RoboDK station: project robotics.rdk

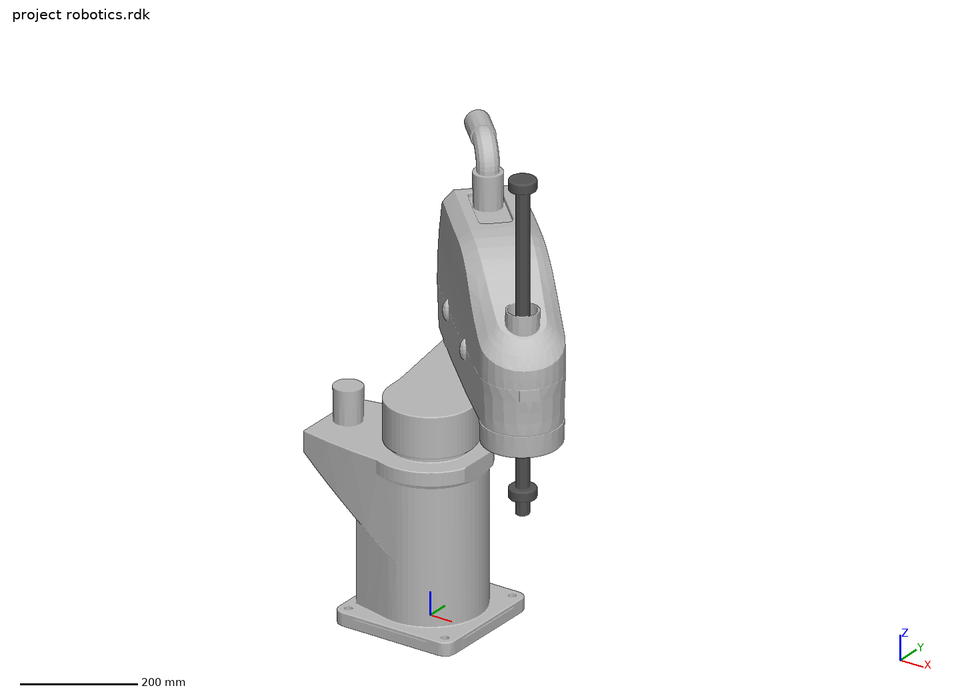
[picture v0: the station drawn from its stored meshes, robots at their saved joint values, targets as dots, program paths as lines]
Station project robotics (saved by RoboDK 5.3.3). Poses are relative to the parent item; angles as X-Y-Z fixed-axis rotations.
  - frame Mitsubishi RH-12SH5535 Base at (0, 0, 0) mm
    - robot Mitsubishi RH-12SH5535: 4 axes, payload 12 kg, reach 600 mm, repeatability 0.03 mm, weight 43 kg
        modified DH rows (alpha deg, a mm, theta deg, d mm): 0, 0, 0, 0; 0, 225, 0, 0; 0, 325, 0, 0 linear; 180, 0, 0, 0
        joint limits [-140, -145, -10, -360] to [140, 145, 340, 360]; home [0, 0, 340, 0]; saved at [99.23, -143.81, 250.69, 0]
  - Python program Prog1 (listed below)

--- Python program Prog1 ---
from robolink import *
from robodk import *

# Start the RoboDK API:
RDK = Robolink()

# Get the robot (first robot found):
robot = RDK.Item('', ITEM_TYPE_ROBOT)
#robot.MoveL([116.40,-80.98,250.69]) #Home
robot.MoveL([99.23,-143.81,250.69])
#MUHD
robot.MoveL([45.01,-116.65,250.69])
robot.MoveL([45.09,-116.72,250.69])
robot.MoveL([47.59,-113.12,250.69])
robot.MoveL([56.09,-127.21,250.69])
robot.MoveL([52.63,-113.23,250.69])
robot.MoveL([63.10,-127.64,250.69])
robot.MoveL([57.81,-112.90,250.69])
robot.MoveL([70.06,-127.43,250.69])
robot.MoveL([67.73,-120.52,250.69])
robot.MoveL([73.23,-126.55,250.69])
robot.MoveL([72.73,-123.86,250.69])
robot.MoveL([70.14,-119.89,250.69])
robot.MoveL([75.68,-125.51,250.69])
robot.MoveL([75.20,-122.42,250.69])
robot.MoveL([65.28,-109.40,250.69])
robot.MoveL([75.24,-122.44,250.69])
robot.MoveL([78.00,-124.57,250.69])
robot.MoveL([73.53,-117.29,250.69])
robot.MoveL([81.10,-123.41,250.69])
robot.MoveL([78.97,-118.82,250.69])
robot.MoveL([76.66,-112.79,250.69])
robot.MoveL([79.05,-118.86,250.69])
robot.MoveL([84.26,-122.47,250.69])
robot.MoveL([79.99,-115.54,250.69])
robot.MoveL([68.82,-103.72,250.69])
robot.MoveL([79.99,-115.51,250.69])
robot.MoveL([86.27,-120.19,250.69])
robot.MoveL([82.62,-115.37,250.69])

#ARIF

#robot.MoveL([92.84,-112.09,250.69])
robot.MoveL([91.16,-119.25,250.69])
robot.MoveL([80.93,-104.10,250.69])
robot.MoveL([87.09,-108.43,250.69])
robot.MoveL([87.25,-116.16,250.69])
robot.MoveL([87.14,-108.48,250.69])
robot.MoveL([92.06,-111.67,250.69])
robot.MoveL([87.22,-105.64,250.69])
robot.MoveL([86.43,-102.87,250.69])
robot.MoveL([90.77,-105.85,250.69])
robot.MoveL([88.73,-102.33,250.69])
robot.MoveL([85.08,-97.90,250.69])
robot.MoveL([88.75,-102.32,250.69])
robot.MoveL([90.10,-102.25,250.69])
robot.MoveL([88.03,-98.47,250.69])
robot.MoveL([79.51,-88.11,250.69])
robot.MoveL([88.21,-98.63,250.69])
robot.MoveL([93.89,-102.15,250.69])
robot.MoveL([92.30,-99.58,250.69])
robot.MoveL([88.33,-96.58,250.69])
robot.MoveL([88.14,-98.49,250.69])
robot.MoveL([88.37,-96.62,250.69])
#robot.MoveL([85.72,-91.70,250.69])
robot.MoveL([87.22,-94.58,250.69])
#robot.MoveL([109.42,-118.65,250.69])

#IKMAL
robot.MoveL([83.51,-88.38,250.69])
robot.MoveL([77.32,-77.82,250.69])
robot.MoveL([79.72,-79.80,250.69])
robot.MoveL([90.90,-91.96,250.69])
robot.MoveL([87.58,-84.52,250.69])
robot.MoveL([74.19,-66.48,250.69])
robot.MoveL([87.60,-84.55,250.69])
robot.MoveL([90.50,-86.45,250.69])
robot.MoveL([83.08,-74.93,250.69])
robot.MoveL([85.58,-76.98,250.69])
robot.MoveL([88.18,-81.99,250.69])
robot.MoveL([89.62,-80.90,250.69])
robot.MoveL([80.65,-67.90,250.69])
robot.MoveL([87.80,-75.54,250.69])
robot.MoveL([78.47,-61.59,250.69])
robot.MoveL([86.05,-70.17,250.69])
robot.MoveL([76.07,-55.33,250.69])
robot.MoveL([83.67,-64.15,250.69])
robot.MoveL([78.17,-54.25,250.69])
robot.MoveL([69.20,-39.81,250.69])
robot.MoveL([78.15,-54.21,250.69])
robot.MoveL([79.37,-53.77,250.69])
robot.MoveL([70.12,-40.01,250.69])
robot.MoveL([76.34,-47.12,250.69])
robot.MoveL([68.59,-35.28,250.69])
robot.MoveL([57.40,-17.69,250.69])
robot.MoveL([50.93,-8.92,250.69])
robot.MoveL([68.71,-35.47,250.69])
robot.MoveL([71.87,-37.60,250.69])
robot.MoveL([66.47,-29.42,250.69])
robot.MoveL([116.40,-80.98,250.69]) #Home
#AB
robot.MoveL([100.54,-139.61,250.69])
robot.MoveL([96.52,-133.61,250.69])
robot.MoveL([93.92,-134.58,250.69])
robot.MoveL([96.52,-133.61,250.69])
robot.MoveL([90.54,-124.22,250.69])
robot.MoveL([99.64,-131.38,250.69])
robot.MoveL([96.61,-133.65,250.69])
robot.MoveL([99.74,-131.46,250.69])
robot.MoveL([106.35,-136.18,250.69])
robot.MoveL([103.42,-131.19,250.69])
robot.MoveL([98.21,-124.67,250.69])
robot.MoveL([93.83,-121.77,250.69])
robot.MoveL([103.32,-131.09,250.69])
robot.MoveL([108.64,-133.92,250.69])
robot.MoveL([105.32,-128.70,250.69])



#GHAFFAR
robot.MoveL([107.70,-126.10,250.69])
robot.MoveL([97.12,-113.94,250.69])
robot.MoveL([100.15,-115.50,250.69])
robot.MoveL([97.15,-113.93,250.69])
robot.MoveL([107.61,-126.08,250.69])
robot.MoveL([106.47,-120.19,250.69])
robot.MoveL([112.57,-126.71,250.69])
robot.MoveL([108.74,-119.49,250.69])
robot.MoveL([97.61,-107.80,250.69])
robot.MoveL([108.80,-119.53,250.69])
robot.MoveL([112.93,-121.18,250.69])
robot.MoveL([106.12,-112.69,250.69])
robot.MoveL([112.93,-118.07,250.69])
robot.MoveL([109.75,-113.65,250.69])
robot.MoveL([105.75,-109.04,250.69])
robot.MoveL([109.83,-113.68,250.69])
robot.MoveL([112.61,-114.73,250.69])
robot.MoveL([106.60,-108.60,250.69])
robot.MoveL([111.73,-111.02,250.69])
robot.MoveL([107.09,-105.54,250.69])
robot.MoveL([95.75,-93.80,250.69])
robot.MoveL([107.08,-105.54,250.69])
robot.MoveL([115.05,-110.92,250.69])
robot.MoveL([111.94,-107.01,250.69])
robot.MoveL([109.83,-105.96,250.69])
robot.MoveL([107.14,-105.54,250.69])
robot.MoveL([109.82,-105.89,250.69])
robot.MoveL([105.75,-100.39,250.69])
robot.MoveL([94.90,-89.40,250.69])
robot.MoveL([105.75,-100.37,250.69])
robot.MoveL([113.10,-105.03,250.69])
robot.MoveL([110.02,-101.16,250.69])
robot.MoveL([107.84,-100.16,250.69])
robot.MoveL([105.72,-100.39,250.69])
robot.MoveL([107.90,-100.21,250.69])
robot.MoveL([105.75,-95.92,250.69])
robot.MoveL([100.60,-88.66,250.69])
robot.MoveL([105.77,-95.97,250.69])
robot.MoveL([108.04,-96.68,250.69])
robot.MoveL([101.83,-88.80,250.69])
robot.MoveL([106.49,-92.52,250.69])
robot.MoveL([103.38,-87.60,250.69])
robot.MoveL([97.80,-81.98,250.69])
robot.MoveL([96.30,-78.14,250.69])
robot.MoveL([102.55,-82.90,250.69])
robot.MoveL([99.21,-78.31,250.69])


robot.MoveL([116.40,-80.98,250.69]) #Home
robot.MoveL([99.23,-143.81,250.69])
robot.RunInstruction('Program_Done')
